    movel(p[0.492326, -0.121867, 0.003000, 0.000000, -3.141593, 0.000000],accel_mss,speed_ms,0,blend_radius_m)
    speed_ms    = 0.050
    movel(p[0.492326, -0.121867, -0.000100, 0.000000, -3.141593, 0.000000],accel_mss,speed_ms,0,blend_radius_m)
    speed_ms    = 0.083
    movel(p[0.490992, -0.123320, -0.000100, 0.000000, -3.141593, 0.000000],accel_mss,speed_ms,0,0.001)
    movel(p[0.489114, -0.124039, -0.000100, 0.000000, -3.141593, 0.000000],accel_mss,speed_ms,0,0.001)
    movel(p[0.487111, -0.123872, -0.000100, 0.000000, -3.141593, 0.000000],accel_mss,speed_ms,0,0.001)
    movel(p[0.485431, -0.122849, -0.000100, 0.000000, -3.141593, 0.000000],accel_mss,speed_ms,0,0.001)
    movel(p[0.484869, -0.122164, -0.000100, 0.000000, -3.141593, 0.000000],accel_mss,speed_ms,0,0.000)
    movel(p[0.484495, -0.121423, -0.000100, 0.000000, -3.141593, 0.000000],accel_mss,speed_ms,0,0.000)
    movel(p[0.484267, -0.120521, -0.000100, 0.000000, -3.141593, 0.000000],accel_mss,speed_ms,0,0.000)
    movel(p[0.484151, -0.119329, -0.000100, 0.000000, -3.141593, 0.000000],accel_mss,speed_ms,0,0.000)
    movel(p[0.484114, -0.118541, -0.000100, 0.000000, -3.141593, 0.000000],accel_mss,speed_ms,0,0.000)
    movel(p[0.484076, -0.117754, -0.000100, 0.000000, -3.141593, 0.000000],accel_mss,speed_ms,0,0.000)
    movel(p[0.483344, -0.117732, -0.000100, 0.000000, -3.141593, 0.000000],accel_mss,speed_ms,0,0.000)
    movel(p[0.482613, -0.117711, -0.000100, 0.000000, -3.141593, 0.000000],accel_mss,speed_ms,0,0.000)
    movel(p[0.481882, -0.117690, -0.000100, 0.000000, -3.141593, 0.000000],accel_mss,speed_ms,0,0.000)
    movel(p[0.481151, -0.117668, -0.000100, 0.000000, -3.141593, 0.000000],accel_mss,speed_ms,0,0.000)
    movel(p[0.481151, -0.117108, -0.000100, 0.000000, -3.141593, 0.000000],accel_mss,speed_ms,0,0.000)
    movel(p[0.481151, -0.116548, -0.000100, 0.000000, -3.141593, 0.000000],accel_mss,speed_ms,0,0.000)
    movel(p[0.481151, -0.115989, -0.000100, 0.000000, -3.141593, 0.000000],accel_mss,speed_ms,0,0.000)
    movel(p[0.481151, -0.115429, -0.000100, 0.000000, -3.141593, 0.000000],accel_mss,speed_ms,0,0.000)
    movel(p[0.483216, -0.115429, -0.000100, 0.000000, -3.141593, 0.000000],accel_mss,speed_ms,0,0.001)
    movel(p[0.485282, -0.115429, -0.000100, 0.000000, -3.141593, 0.000000],accel_mss,speed_ms,0,0.001)
    movel(p[0.487348, -0.115429, -0.000100, 0.000000, -3.141593, 0.000000],accel_mss,speed_ms,0,0.001)
    movel(p[0.489414, -0.115429, -0.000100, 0.000000, -3.141593, 0.000000],accel_mss,speed_ms,0,0.001)
    movel(p[0.489392, -0.115973, -0.000100, 0.000000, -3.141593, 0.000000],accel_mss,speed_ms,0,0.000)
    movel(p[0.489370, -0.116516, -0.000100, 0.000000, -3.141593, 0.000000],accel_mss,speed_ms,0,0.000)
    movel(p[0.489348, -0.117060, -0.000100, 0.000000, -3.141593, 0.000000],accel_mss,speed_ms,0,0.000)
    movel(p[0.489326, -0.117604, -0.000100, 0.000000, -3.141593, 0.000000],accel_mss,speed_ms,0,0.000)
    movel(p[0.488587, -0.117625, -0.000100, 0.000000, -3.141593, 0.000000],accel_mss,speed_ms,0,0.000)
    movel(p[0.487849, -0.117647, -0.000100, 0.000000, -3.141593, 0.000000],accel_mss,speed_ms,0,0.000)
    movel(p[0.487111, -0.117669, -0.000100, 0.000000, -3.141593, 0.000000],accel_mss,speed_ms,0,0.000)
    movel(p[0.486373, -0.117690, -0.000100, 0.000000, -3.141593, 0.000000],accel_mss,speed_ms,0,0.000)
    movel(p[0.486399, -0.118431, -0.000100, 0.000000, -3.141593, 0.000000],accel_mss,speed_ms,0,0.000)
    movel(p[0.486424, -0.119173, -0.000100, 0.000000, -3.141593, 0.000000],accel_mss,speed_ms,0,0.000)
    movel(p[0.486466, -0.120042, -0.000100, 0.000000, -3.141593, 0.000000],accel_mss,speed_ms,0,0.000)
    movel(p[0.486528, -0.120480, -0.000100, 0.000000, -3.141593, 0.000000],accel_mss,speed_ms,0,0.000)
    movel(p[0.486644, -0.120777, -0.000100, 0.000000, -3.141593, 0.000000],accel_mss,speed_ms,0,0.000)
    movel(p[0.486851, -0.121056, -0.000100, 0.000000, -3.141593, 0.000000],accel_mss,speed_ms,0,0.000)
    movel(p[0.487734, -0.121682, -0.000100, 0.000000, -3.141593, 0.000000],accel_mss,speed_ms,0,0.000)
    movel(p[0.488735, -0.121857, -0.000100, 0.000000, -3.141593, 0.000000],accel_mss,speed_ms,0,0.000)
    movel(p[0.489671, -0.121545, -0.000100, 0.000000, -3.141593, 0.000000],accel_mss,speed_ms,0,0.000)
    movel(p[0.490376, -0.120812, -0.000100, 0.000000, -3.141593, 0.000000],accel_mss,speed_ms,0,0.000)
    movel(p[0.490547, -0.120370, -0.000100, 0.000000, -3.141593, 0.000000],accel_mss,speed_ms,0,0.000)
    movel(p[0.490637, -0.119732, -0.000100, 0.000000, -3.141593, 0.000000],accel_mss,speed_ms,0,0.000)
    movel(p[0.490686, -0.118629, -0.000100, 0.000000, -3.141593, 0.000000],accel_mss,speed_ms,0,0.000)
    movel(p[0.490722, -0.116059, -0.000100, 0.000000, -3.141593, 0.000000],accel_mss,speed_ms,0,blend_radius_m)
    movel(p[0.490758, -0.113259, -0.000100, 0.000000, -3.141593, 0.000000],accel_mss,speed_ms,0,blend_radius_m)
    movel(p[0.490804, -0.112342, -0.000100, 0.000000, -3.141593, 0.000000],accel_mss,speed_ms,0,0.000)
    movel(p[0.490899, -0.111894, -0.000100, 0.000000, -3.141593, 0.000000],accel_mss,speed_ms,0,0.000)
    movel(p[0.491097, -0.111689, -0.000100, 0.000000, -3.141593, 0.000000],accel_mss,speed_ms,0,0.000)
    movel(p[0.491268, -0.111600, -0.000100, 0.000000, -3.141593, 0.000000],accel_mss,speed_ms,0,0.000)
    movel(p[0.491540, -0.111413, -0.000100, 0.000000, -3.141593, 0.000000],accel_mss,speed_ms,0,0.000)
    movel(p[0.491846, -0.111179, -0.000100, 0.000000, -3.141593, 0.000000],accel_mss,speed_ms,0,0.000)
    movel(p[0.492145, -0.110926, -0.000100, 0.000000, -3.141593, 0.000000],accel_mss,speed_ms,0,0.000)
    movel(p[0.492505, -0.110609, -0.000100, 0.000000, -3.141593, 0.000000],accel_mss,speed_ms,0,0.000)
    movel(p[0.492865, -0.110291, -0.000100, 0.000000, -3.141593, 0.000000],accel_mss,speed_ms,0,0.000)
    movel(p[0.492843, -0.112982, -0.000100, 0.000000, -3.141593, 0.000000],accel_mss,speed_ms,0,blend_radius_m)
    movel(p[0.492820, -0.115672, -0.000100, 0.000000, -3.141593, 0.000000],accel_mss,speed_ms,0,blend_radius_m)
    movel(p[0.492798, -0.118363, -0.000100, 0.000000, -3.141593, 0.000000],accel_mss,speed_ms,0,blend_radius_m)
    movel(p[0.492776, -0.121054, -0.000100, 0.000000, -3.141593, 0.000000],accel_mss,speed_ms,0,blend_radius_m)
    movel(p[0.492551, -0.121460, -0.000100, 0.000000, -3.141593, 0.000000],accel_mss,speed_ms,0,0.000)
    movel(p[0.492326, -0.121867, -0.000100, 0.000000, -3.141593, 0.000000],accel_mss,speed_ms,0,0.000)
    speed_ms    = 0.050
    movel(p[0.492326, -0.121867, 0.003000, 0.000000, -3.141593, 0.000000],accel_mss,speed_ms,0,blend_radius_m)
    speed_ms    = 1.000
    movel(p[0.492326, -0.121867, 0.015000, 0.000000, -3.141593, 0.000000],accel_mss,speed_ms,0,blend_radius_m)

    movel(p[0.502602, -0.114608, 0.015000, 0.000000, -3.141593, 0.000000],accel_mss,speed_ms,0,blend_radius_m)

    movel(p[0.502602, -0.114608, 0.003000, 0.000000, -3.141593, 0.000000],accel_mss,speed_ms,0,blend_radius_m)
    speed_ms    = 0.050
    movel(p[0.502602, -0.114608, -0.000100, 0.000000, -3.141593, 0.000000],accel_mss,speed_ms,0,blend_radius_m)
    speed_ms    = 0.083
    movel(p[0.502864, -0.114345, -0.000100, 0.000000, -3.141593, 0.000000],accel_mss,speed_ms,0,0.000)
    movel(p[0.503127, -0.114082, -0.000100, 0.000000, -3.141593, 0.000000],accel_mss,speed_ms,0,0.000)
    movel(p[0.503390, -0.113820, -0.000100, 0.000000, -3.141593, 0.000000],accel_mss,speed_ms,0,0.000)
    movel(p[0.503653, -0.113557, -0.000100, 0.000000, -3.141593, 0.000000],accel_mss,speed_ms,0,0.000)
    movel(p[0.505158, -0.115062, -0.000100, 0.000000, -3.141593, 0.000000],accel_mss,speed_ms,0,0.001)
    movel(p[0.506663, -0.116568, -0.000100, 0.000000, -3.141593, 0.000000],accel_mss,speed_ms,0,0.001)
    movel(p[0.508169, -0.118073, -0.000100, 0.000000, -3.141593, 0.000000],accel_mss,speed_ms,0,0.001)
    movel(p[0.509674, -0.119578, -0.000100, 0.000000, -3.141593, 0.000000],accel_mss,speed_ms,0,0.001)
    movel(p[0.509474, -0.119816, -0.000100, 0.000000, -3.141593, 0.000000],accel_mss,speed_ms,0,0.000)
    movel(p[0.509274, -0.120054, -0.000100, 0.000000, -3.141593, 0.000000],accel_mss,speed_ms,0,0.000)
    movel(p[0.509108, -0.120236, -0.000100, 0.000000, -3.141593, 0.000000],accel_mss,speed_ms,0,0.000)
    movel(p[0.508941, -0.120389, -0.000100, 0.000000, -3.141593, 0.000000],accel_mss,speed_ms,0,0.000)
    movel(p[0.508792, -0.120501, -0.000100, 0.000000, -3.141593, 0.000000],accel_mss,speed_ms,0,0.000)
    movel(p[0.508585, -0.120483, -0.000100, 0.000000, -3.141593, 0.000000],accel_mss,speed_ms,0,0.000)
    movel(p[0.507709, -0.119659, -0.000100, 0.000000, -3.141593, 0.000000],accel_mss,speed_ms,0,0.000)
    movel(p[0.506713, -0.118703, -0.000100, 0.000000, -3.141593, 0.000000],accel_mss,speed_ms,0,0.001)
    movel(p[0.505565, -0.117568, -0.000100, 0.000000, -3.141593, 0.000000],accel_mss,speed_ms,0,0.001)
    movel(p[0.504083, -0.116088, -0.000100, 0.000000, -3.141593, 0.000000],accel_mss,speed_ms,0,0.001)
    movel(p[0.502602, -0.114608, -0.000100, 0.000000, -3.141593, 0.000000],accel_mss,speed_ms,0,0.001)
    speed_ms    = 0.050
    movel(p[0.502602, -0.114608, 0.003000, 0.000000, -3.141593, 0.000000],accel_mss,speed_ms,0,blend_radius_m)
    speed_ms    = 1.000
    movel(p[0.502602, -0.114608, 0.015000, 0.000000, -3.141593, 0.000000],accel_mss,speed_ms,0,blend_radius_m)

    movel(p[0.506318, -0.113033, 0.015000, 0.000000, -3.141593, 0.000000],accel_mss,speed_ms,0,blend_radius_m)

    movel(p[0.506318, -0.113033, 0.003000, 0.000000, -3.141593, 0.000000],accel_mss,speed_ms,0,blend_radius_m)
    speed_ms    = 0.050
    movel(p[0.506318, -0.113033, -0.000100, 0.000000, -3.141593, 0.000000],accel_mss,speed_ms,0,blend_radius_m)
    speed_ms    = 0.083
    movel(p[0.506196, -0.112240, -0.000100, 0.000000, -3.141593, 0.000000],accel_mss,speed_ms,0,0.000)
    movel(p[0.506287, -0.111464, -0.000100, 0.000000, -3.141593, 0.000000],accel_mss,speed_ms,0,0.000)
    movel(p[0.506588, -0.110660, -0.000100, 0.000000, -3.141593, 0.000000],accel_mss,speed_ms,0,0.000)
    movel(p[0.507392, -0.109520, -0.000100, 0.000000, -3.141593, 0.000000],accel_mss,speed_ms,0,0.001)
    movel(p[0.508467, -0.108736, -0.000100, 0.000000, -3.141593, 0.000000],accel_mss,speed_ms,0,0.001)
    movel(p[0.509654, -0.108414, -0.000100, 0.000000, -3.141593, 0.000000],accel_mss,speed_ms,0,0.000)
    movel(p[0.510787, -0.108599, -0.000100, 0.000000, -3.141593, 0.000000],accel_mss,speed_ms,0,0.000)
    movel(p[0.511124, -0.108751, -0.000100, 0.000000, -3.141593, 0.000000],accel_mss,speed_ms,0,0.000)
    movel(p[0.511218, -0.108847, -0.000100, 0.000000, -3.141593, 0.000000],accel_mss,speed_ms,0,0.000)
    movel(p[0.511219, -0.108975, -0.000100, 0.000000, -3.141593, 0.000000],accel_mss,speed_ms,0,0.000)
    movel(p[0.511083, -0.109264, -0.000100, 0.000000, -3.141593, 0.000000],accel_mss,speed_ms,0,0.000)
    movel(p[0.510856, -0.109630, -0.000100, 0.000000, -3.141593, 0.000000],accel_mss,speed_ms,0,0.000)
    movel(p[0.510631, -0.109820, -0.000100, 0.000000, -3.141593, 0.000000],accel_mss,speed_ms,0,0.000)
    movel(p[0.510314, -0.109911, -0.000100, 0.000000, -3.141593, 0.000000],accel_mss,speed_ms,0,0.000)
    movel(p[0.509736, -0.109945, -0.000100, 0.000000, -3.141593, 0.000000],accel_mss,speed_ms,0,0.000)
    movel(p[0.509395, -0.109969, -0.000100, 0.000000, -3.141593, 0.000000],accel_mss,speed_ms,0,0.000)
    movel(p[0.509071, -0.110028, -0.000100, 0.000000, -3.141593, 0.000000],accel_mss,speed_ms,0,0.000)
    movel(p[0.508788, -0.110117, -0.000100, 0.000000, -3.141593, 0.000000],accel_mss,speed_ms,0,0.000)
    movel(p[0.508570, -0.110231, -0.000100, 0.000000, -3.141593, 0.000000],accel_mss,speed_ms,0,0.000)
    movel(p[0.508168, -0.110618, -0.000100, 0.000000, -3.141593, 0.000000],accel_mss,speed_ms,0,0.000)
    movel(p[0.507830, -0.111196, -0.000100, 0.000000, -3.141593, 0.000000],accel_mss,speed_ms,0,0.000)
    movel(p[0.507622, -0.111818, -0.000100, 0.000000, -3.141593, 0.000000],accel_mss,speed_ms,0,0.000)
    movel(p[0.507613, -0.112337, -0.000100, 0.000000, -3.141593, 0.000000],accel_mss,speed_ms,0,0.000)
    movel(p[0.507824, -0.112949, -0.000100, 0.000000, -3.141593, 0.000000],accel_mss,speed_ms,0,0.000)
    movel(p[0.508250, -0.113628, -0.000100, 0.000000, -3.141593, 0.000000],accel_mss,speed_ms,0,0.000)
    movel(p[0.508819, -0.114285, -0.000100, 0.000000, -3.141593, 0.000000],accel_mss,speed_ms,0,0.000)
    movel(p[0.509467, -0.114832, -0.000100, 0.000000, -3.141593, 0.000000],accel_mss,speed_ms,0,0.000)
    movel(p[0.509928, -0.115141, -0.000100, 0.000000, -3.141593, 0.000000],accel_mss,speed_ms,0,0.000)
    movel(p[0.510271, -0.115314, -0.000100, 0.000000, -3.141593, 0.000000],accel_mss,speed_ms,0,0.000)
    movel(p[0.510597, -0.115400, -0.000100, 0.000000, -3.141593, 0.000000],accel_mss,speed_ms,0,0.000)
    movel(p[0.510988, -0.115428, -0.000100, 0.000000, -3.141593, 0.000000],accel_mss,speed_ms,0,0.000)
    movel(p[0.511871, -0.115265, -0.000100, 0.000000, -3.141593, 0.000000],accel_mss,speed_ms,0,0.000)
    movel(p[0.512570, -0.114801, -0.000100, 0.000000, -3.141593, 0.000000],accel_mss,speed_ms,0,0.000)
    movel(p[0.512984, -0.114101, -0.000100, 0.000000, -3.141593, 0.000000],accel_mss,speed_ms,0,0.000)
    movel(p[0.513059, -0.113267, -0.000100, 0.000000, -3.141593, 0.000000],accel_mss,speed_ms,0,0.000)
    movel(p[0.513023, -0.113015, -0.000100, 0.000000, -3.141593, 0.000000],accel_mss,speed_ms,0,0.000)
    movel(p[0.512978, -0.112766, -0.000100, 0.000000, -3.141593, 0.000000],accel_mss,speed_ms,0,0.000)
    movel(p[0.512930, -0.112550, -0.000100, 0.000000, -3.141593, 0.000000],accel_mss,speed_ms,0,0.000)
    movel(p[0.512888, -0.112421, -0.000100, 0.000000, -3.141593, 0.000000],accel_mss,speed_ms,0,0.000)
    movel(p[0.512878, -0.112300, -0.000100, 0.000000, -3.141593, 0.000000],accel_mss,speed_ms,0,0.000)
    movel(p[0.512939, -0.112184, -0.000100, 0.000000, -3.141593, 0.000000],accel_mss,speed_ms,0,0.000)
    movel(p[0.513083, -0.112065, -0.000100, 0.000000, -3.141593, 0.000000],accel_mss,speed_ms,0,0.000)
    movel(p[0.513326, -0.111934, -0.000100, 0.000000, -3.141593, 0.000000],accel_mss,speed_ms,0,0.000)
    movel(p[0.513826, -0.111724, -0.000100, 0.000000, -3.141593, 0.000000],accel_mss,speed_ms,0,0.000)
    movel(p[0.514091, -0.111716, -0.000100, 0.000000, -3.141593, 0.000000],accel_mss,speed_ms,0,0.000)
    movel(p[0.514271, -0.111866, -0.000100, 0.000000, -3.141593, 0.000000],accel_mss,speed_ms,0,0.000)
    movel(p[0.514427, -0.112259, -0.000100, 0.000000, -3.141593, 0.000000],accel_mss,speed_ms,0,0.000)
    movel(p[0.514594, -0.113173, -0.000100, 0.000000, -3.141593, 0.000000],accel_mss,speed_ms,0,0.000)
    movel(p[0.514523, -0.113998, -0.000100, 0.000000, -3.141593, 0.000000],accel_mss,speed_ms,0,0.000)
    movel(p[0.514200, -0.114782, -0.000100, 0.000000, -3.141593, 0.000000],accel_mss,speed_ms,0,0.000)
    movel(p[0.513613, -0.115573, -0.000100, 0.000000, -3.141593, 0.000000],accel_mss,speed_ms,0,0.000)
    movel(p[0.512987, -0.116165, -0.000100, 0.000000, -3.141593, 0.000000],accel_mss,speed_ms,0,0.000)
    movel(p[0.512359, -0.116554, -0.000100, 0.000000, -3.141593, 0.000000],accel_mss,speed_ms,0,0.000)
    movel(p[0.511668, -0.116771, -0.000100, 0.000000, -3.141593, 0.000000],accel_mss,speed_ms,0,0.000)
    movel(p[0.510851, -0.116843, -0.000100, 0.000000, -3.141593, 0.000000],accel_mss,speed_ms,0,0.000)
    movel(p[0.510350, -0.116824, -0.000100, 0.000000, -3.141593, 0.000000],accel_mss,speed_ms,0,0.000)
    movel(p[0.509945, -0.116767, -0.000100, 0.000000, -3.141593, 0.000000],accel_mss,speed_ms,0,0.000)
    movel(p[0.509583, -0.116661, -0.000100, 0.000000, -3.141593, 0.000000],accel_mss,speed_ms,0,0.000)
    movel(p[0.509217, -0.116497, -0.000100, 0.000000, -3.141593, 0.000000],accel_mss,speed_ms,0,0.000)
    movel(p[0.508473, -0.116018, -0.000100, 0.000000, -3.141593, 0.000000],accel_mss,speed_ms,0,0.000)
    movel(p[0.507748, -0.115372, -0.000100, 0.000000, -3.141593, 0.000000],accel_mss,speed_ms,0,0.000)
    movel(p[0.507116, -0.114636, -0.000100, 0.000000, -3.141593, 0.000000],accel_mss,speed_ms,0,0.000)
    movel(p[0.506653, -0.113887, -0.000100, 0.000000, -3.141593, 0.000000],accel_mss,speed_ms,0,0.000)
    movel(p[0.506318, -0.113033, -0.000100, 0.000000, -3.141593, 0.000000],accel_mss,speed_ms,0,0.000)
    speed_ms    = 0.050
    movel(p[0.506318, -0.113033, 0.003000, 0.000000, -3.141593, 0.000000],accel_mss,speed_ms,0,blend_radius_m)
    speed_ms    = 1.000
    movel(p[0.506318, -0.113033, 0.015000, 0.000000, -3.141593, 0.000000],accel_mss,speed_ms,0,blend_radius_m)

    movel(p[0.514600, -0.147080, 0.015000, 0.000000, -3.141593, 0.000000],accel_mss,speed_ms,0,blend_radius_m)
    movel(p[0.514600, -0.147080, 0.115000, 0.000000, -3.141593, 0.000000],accel_mss,speed_ms,0,blend_radius_m)

  $ 3 "Halt"
  halt
end
